// TIA Portal V20 export
DATA_BLOCK "TEST"   // DB207
// stored: MemoryReserve 100, Namespace Unit1.Em5
   VAR RETAIN
      bit : Array[0..19] of Bool;
      Dummy : Array[0..63] of Bool;
   END_VAR
BEGIN
END_DATA_BLOCK
